// Automatisch erzeugter Code: NICHT EDITIEREN
FUNCTION CheckRangeSigned : DINT
VAR_INPUT
	value, lower, upper: DINT;
END_VAR

// Automatisch erzeugter Code: Es handelt sich hierbei um einen Implementierungsvorschlag.
{noflow}
IF (value < lower) THEN
	CheckRangeSigned := lower;
ELSIF(value > upper) THEN
	CheckRangeSigned := upper;
ELSE
	CheckRangeSigned := value;
END_IF
{flow}

END_FUNCTION

(* stored: Version 1.1.0.1, ProductVersion 3.1.4024.10
   POU CheckRangeSigned: Id {0da657b8-70db-4c6f-94b3-717711f9d839}, SpecialFunc CheckRangeSigned *)
